(* IEC 61131-3 sources: Laboratorijsko-busace-postrojenje/Logging/read_data, 2 files *)

(* ---- read_data.st ---- *)
(********************************************************************
 * COPYRIGHT -- Bernecker + Rainer
 ********************************************************************
 * Program: read_data
 * File: read_data.st
 * Author: Bernecker & Rainer
 * Created: April 20, 2009
 ********************************************************************
 * Implementation of program read_data
 ********************************************************************)

PROGRAM _INIT

	step := WAIT;

END_PROGRAM

PROGRAM _CYCLIC

CASE step OF

	WAIT:

		IF start_reading_usb_data = TRUE THEN
			step := CREATE_NODE_ID_LIST;  (*start FUBs below*)
		ELSE
			step := WAIT;
		END_IF;

	CREATE_NODE_ID_LIST:  (*Library AsUSB - Functionblock USBNodeListGet()*)

		UsbNodeListGet_0.enable := 1;
		UsbNodeListGet_0.pBuffer := ADR(node_id_buffer);  (*pointer to buffer - UDINT array is assigned*)
		UsbNodeListGet_0.bufferSize := SIZEOF(node_id_buffer);  (*size of node-id-buffer-array*)
		UsbNodeListGet_0.filterInterfaceClass := asusb_CLASS_MASS_STORAGE;  (*filter on mass storage devices is set*)
		UsbNodeListGet_0.filterInterfaceSubClass := 0;  (*no filer is set*)
		UsbNodeListGet_0;

		IF UsbNodeListGet_0.status = 0 THEN
        	step := READ_DEVICE_DATA;  (*FUB worked correctly => next step*)
		ELSIF UsbNodeListGet_0.status = ERR_FUB_BUSY THEN
			step := CREATE_NODE_ID_LIST;  (*FUB work asynchron => called until status isn't BUSY*)
		ELSE
			step := ERROR_CASE;  (*error occured*)
		END_IF;

	READ_DEVICE_DATA:  (*Library AsUSB - Functionblock USBNodeGet()*)

		UsbNodeGet_0.enable := 1;
		UsbNodeGet_0.nodeId := node_id_buffer[node];  (*specific node is read out of node_id_buffer*)
		UsbNodeGet_0.pBuffer := ADR(usb_data_buffer[node]);  (*data of specific node get stored in usb_data_buffer*)
		UsbNodeGet_0.bufferSize := SIZEOF (usb_data_buffer[node]);  (*size of specific node is read out usb_data_buffer*)
		UsbNodeGet_0;

		IF UsbNodeGet_0.status = 0 THEN  (*FUB worked correctly*)
			node := node + 1;  (*next node to be read out of buffer*)
			IF node = UsbNodeListGet_0.listNodes THEN  (*last existing node is reached*)
				node := 0;
				step := GET_DESCRIPTOR;  (*all nodes are read out of buffer*)
			END_IF;

		ELSIF UsbNodeGet_0.status = ERR_FUB_BUSY THEN
			step := READ_DEVICE_DATA;  (*FUB work asynchron => called until status isn't BUSY*)
		ELSE
			step := ERROR_CASE;  (*error occured*)
		END_IF;

	GET_DESCRIPTOR:  (*Library AsUSB - Functionblock USBDescriptorGet()*)

		UsbDescriptorGet_0.enable := 1;
		UsbDescriptorGet_0.nodeId := node_id_buffer[node];  (*specific node is read out of node_id_buffer*)
		UsbDescriptorGet_0.requestType := 0;  (*Request for device*)
        UsbDescriptorGet_0.descriptorType := 1;  (*Determines the device descriptor*)
		UsbDescriptorGet_0.languageId := 0;  (*for device and configuration descriptors*)
		UsbDescriptorGet_0.pBuffer := ADR(device_descriptor[node]);  (*descriptor-data of specific node get stored in device_descriptor-buffer*)
		UsbDescriptorGet_0.bufferSize := SIZEOF(device_descriptor[node]);  (*size of specific node is read out device_descriptor-buffer*)
		UsbDescriptorGet_0;

		IF UsbDescriptorGet_0.status = 0 THEN  (*FUB worked correctly*)
			node := node + 1;  (*next node to be read out of buffer*)
			IF node = UsbNodeListGet_0.listNodes THEN  (*last existing node is reached*)
				node := 0;
				step := CREATE_FILE_DEVICE;  (*all nodes are read out of buffer*)
			END_IF;

		ELSIF UsbDescriptorGet_0.status = ERR_FUB_BUSY THEN
			step := GET_DESCRIPTOR;  (*FUB work asynchron => called until status isn't BUSY*)
		ELSE
			step := ERROR_CASE;  (*error occured*)
		END_IF;

	CREATE_FILE_DEVICE:  (*Library FileIO - Functionblock DevLink() - create file out of data just from 1. USB*)

		strcpy(ADR(device_name), ADR('DEVICE1'));  (*fixed Device-Name get copied to device_name-Variable*)
		strcpy(ADR(device_param), ADR('/DEVICE='));  (*first part of parameter get copied to device_param-Variable*)
		strcat(ADR(device_param), ADR(usb_data_buffer[0].ifName));  (*second part get added to device_param-Variable*)

		DevLink_0.enable := 1;
		DevLink_0.pDevice := ADR(device_name);  (*Devicename is assigned*)
		DevLink_0.pParam := ADR(device_param);  (*the path of the Device is assigned*)
		DevLink_0;

		IF DevLink_0.status = 0 THEN
			step := DIRECTORY_INFO;  (*FUB worked correctly => next step*)
		ELSIF DevLink_0.status = ERR_FUB_BUSY THEN
			step := CREATE_FILE_DEVICE;  (*FUB work asynchron => called until status isn't BUSY*)
		ELSE
			step := ERROR_CASE;  (*error occured*)
		END_IF;

	DIRECTORY_INFO:  (*Library FileIO - Functionblock DirInfo()*)

		DirInfo_0.enable := 1;
		DirInfo_0.pDevice := ADR(device_name);  (*Devicename is assigned*)
		DirInfo_0.pPath := 0;  (*no path is needed => value = 0*)
		DirInfo_0;

		IF DirInfo_0.status = 0 THEN
			step := DIRECTORY_READ;  (*FUB worked correctly => next step*)
		ELSIF DirInfo_0.status = ERR_FUB_BUSY THEN
			step := DIRECTORY_INFO;  (*FUB work asynchron => called until status isn't BUSY*)
		ELSE
			step := ERROR_CASE;  (*error occured*)
		END_IF;

	DIRECTORY_READ:  (*Library FileIO - Functionblock DirRead()*)

		DirRead_0.enable := 1;
		DirRead_0.pDevice := ADR(device_name);  (*Devicename is assigned*)
		DirRead_0.pPath := 0;  (*no path is needed => value = 0*)
		DirRead_0.entry := 1;  (*only the first entry is read out*)
		DirRead_0.option := fiBOTH;  (*Collect information from files and directories*)
		DirRead_0.pData := ADR(device_data);  (*device_data-variable with fiDIR_READ_DATA type is assigned to data-buffer*)
		DirRead_0.data_len := SIZEOF(device_data); (*size of device_data-variable is read out*)
		DirRead_0;

		IF DirRead_0.status = 0 THEN
				(*step := UNLINK_DEVICE;*)  (*FUB worked correctly => next step*)
				step := WAIT;
		ELSIF DirRead_0.status = ERR_FUB_BUSY THEN
			step := DIRECTORY_READ;  (*FUB work asynchron => called until status isn't BUSY*)
		ELSE
			step := ERROR_CASE;  (*error occured*)
		END_IF;

	UNLINK_DEVICE:  (*Library FileIO - Functionblock DevUnlink()*)

		DevUnlink_0.enable := 1;
		DevUnlink_0.handle := DevLink_0.handle;  (*handle from DevLink is assigned to cut the connection to specific file-device*)
		DevUnlink_0;

		IF DevUnlink_0.status = 0 THEN
			step := FINISH;  (*FUB worked correctly => next step*)
		ELSIF DevUnlink_0.status = ERR_FUB_BUSY THEN
			step := UNLINK_DEVICE;  (*FUB work asynchron => called until status isn't BUSY*)
		ELSE
			step := ERROR_CASE;  (*error occured*)
		END_IF;

	FINISH:  (*successfully finished*)

		start_reading_usb_data := FALSE;
		step := WAIT;  (*back to beginning - wait for start_reading_usb_data to be set*)

	ERROR_CASE:	(*error-handling*)

END_CASE;

END_PROGRAM

(* ---- read_data.var ---- *)
(********************************************************************
 * COPYRIGHT -- Bernecker + Rainer
 ********************************************************************
 * Program: read_data
 * File: read_data.var
 * Author: Bernecker & Rainer
 * Created: April 20, 2009
 ********************************************************************
 * Local variables of program read_data
 ********************************************************************)
VAR CONSTANT
	CREATE_NODE_ID_LIST : USINT := 2; (*Function step: Create a list of Node-IDs from all active USB devices*)
	READ_DEVICE_DATA : USINT := 3; (*Function step: Read out the specific data from the Node-IDs*)
	GET_DESCRIPTOR : USINT := 4; (*Function step: Read out the descriptor data from the Node-IDs*)
	CREATE_FILE_DEVICE : USINT := 5; (*Function step: Create file out of data from USB device*)
	DIRECTORY_READ : USINT := 7; (*Function step: Read out to data from linked File Device*)
	UNLINK_DEVICE : USINT := 9; (*Function step: Unlink the File Device from specific path*)
	FINISH : USINT := 8; (*Function step: Function chain is finished - back to WAIT*)
	WAIT : USINT := 0; (*Function step: Wait for starting the Function chain*)
	DIRECTORY_INFO : USINT := 6; (*Function step: Read out the Info about the connected File Device*)
	ERROR_CASE : USINT := 1; (*Function step: Jump to this step in every case of Error occuring in the Function chain*)
END_VAR
VAR
	device_data : fiDIR_READ_DATA := (0); (*Buffer to store device data*)
	device_descriptor : ARRAY[0..4] OF usbDeviceDescr_typ; (*Buffer to store descriptor data of device*)
	usb_data_buffer : ARRAY[0..4] OF usbNode_typ; (*Defined data_typ of AsUSB - Library*)
	node_id_buffer : ARRAY[0..4] OF UDINT; (*Different nodeIDs saved in array-elements*)
	UsbNodeListGet_0 : UsbNodeListGet; (*Type of FUB UsbNodeListGet*)
	step : USINT; (*Determines the Function step*)
	UsbNodeGet_0 : UsbNodeGet; (*Type of FUB UsbNodeGet*)
	start_reading_usb_data : BOOL := TRUE; (*If TRUE - Function chain gets started*)
	node : USINT; (*Node number*)
	DevLink_0 : DevLink; (*Type of FUB DevLink*)
	UsbDescriptorGet_0 : UsbDescriptorGet; (*Type of FUB UsbDescriptorGet*)
	device_name : STRING[80]; (*Name of the USB device - optional *)
	device_param : STRING[80]; (*Connection path of USB device*)
	DirInfo_0 : DirInfo; (*Type of FUB DirInfo*)
	DirRead_0 : DirRead; (*Type of FUB DirRead*)
	DevUnlink_0 : DevUnlink; (*Type of FUB DevUnlink*)
END_VAR
